(* IEC 61131-3 sources: sigmatek-logger-api/IXON_API/Class/Pulse, 1 file *)

(* ---- Pulse.st ---- *)
(*!
<Class
	Name               = "Pulse"
	Revision           = "0.0"
	RealtimeTask       = "false"
	CyclicTask         = "true"
	DefCyclictime      = "500 ms"
	BackgroundTask     = "false"
	Sigmatek           = "false"
	OSInterface        = "false"
	HighPriority       = "false"
	Automatic          = "false"
	UpdateMode         = "Prescan"
	SharedCommandTable = "true"
	Objectsize         = "(284,120)">
	<Channels>
		<Server Name="ClassSvr" Visualized="false" Initialize="false" WriteProtected="true" Retentive="false"/>
		<Client Name="PulseOut1" Required="true" Internal="false"/>
		<Client Name="PulseOut2" Required="true" Internal="false"/>
		<Client Name="PulseOut3" Required="true" Internal="false"/>
	</Channels>
</Class>
*)
Pulse : CLASS
  //Servers:
	ClassSvr 	: SvrChCmd_DINT;
  //Clients:
	PulseOut1 	: CltCh_DINT;
	PulseOut2 	: CltCh_DINT;
	PulseOut3 	: CltCh_DINT;
  //Variables:
  //Functions:

	FUNCTION VIRTUAL GLOBAL CyWork
		VAR_INPUT
			EAX 	: UDINT;
		END_VAR
		VAR_OUTPUT
			state (EAX) 	: UDINT;
		END_VAR;
  //Tables:
	FUNCTION @STD
		VAR_OUTPUT
			ret_code	: CONFSTATES;
		END_VAR;
	FUNCTION GLOBAL TAB @CT_;
END_CLASS;

FUNCTION VIRTUAL GLOBAL Pulse::CyWork
	VAR_INPUT
		EAX 	: UDINT;
	END_VAR
	VAR_OUTPUT
		state (EAX) 	: UDINT;
	END_VAR

	state := READY;

  PulseOut1 := PulseOut1 + 1;
  PulseOut1.Write(input:=PulseOut1);

  PulseOut2 := PulseOut2 + 1;
  PulseOut2.Write(input:=PulseOut2);
  PulseOut3.Write(input:=PulseOut2);
END_FUNCTION
